// TIA Portal V19 export
TYPE "ItemInfo_UDT"
   STRUCT
      LocateActive : Bool;
      TrippedInd : Bool;
      IsolatedInd : Bool;
      VSD_Fault : Bool;
      VSD_Alarm : Bool;
      sv_3Activated : Bool;
      fb_error : Bool;   // Alarm feedback error
      sv_2Activated : Bool;
      activated : Bool;
      changing : Bool;
      faulty : Bool;
      auto_man : Bool;   // Manual = 1
      man_on_off : Bool;
      Reset_FB : Bool;
      ManualSelected : Bool;
      Set_FB : Bool;
   END_STRUCT;
END_TYPE
